{attribute 'TcGenerated'}
{attribute 'no-analysis'}
{attribute 'linkalways'}
// This function has been automatically generated from the project information.
VAR_GLOBAL CONSTANT
	{attribute 'const_non_replaced'}
	stLibVersion_RS485_Hausbus_Kernal : ST_LibVersion := (iMajor := 1, iMinor := 4, iBuild := 7, iRevision := 0, nFlags := 1, sVersion := '1.4.7');
END_VAR

(* stored: Version 1.1.0.1, ProductVersion 3.1.4024.16
   GVL Global_Version: Id {6c393c68-e974-4352-926f-7cff922213c9} *)
